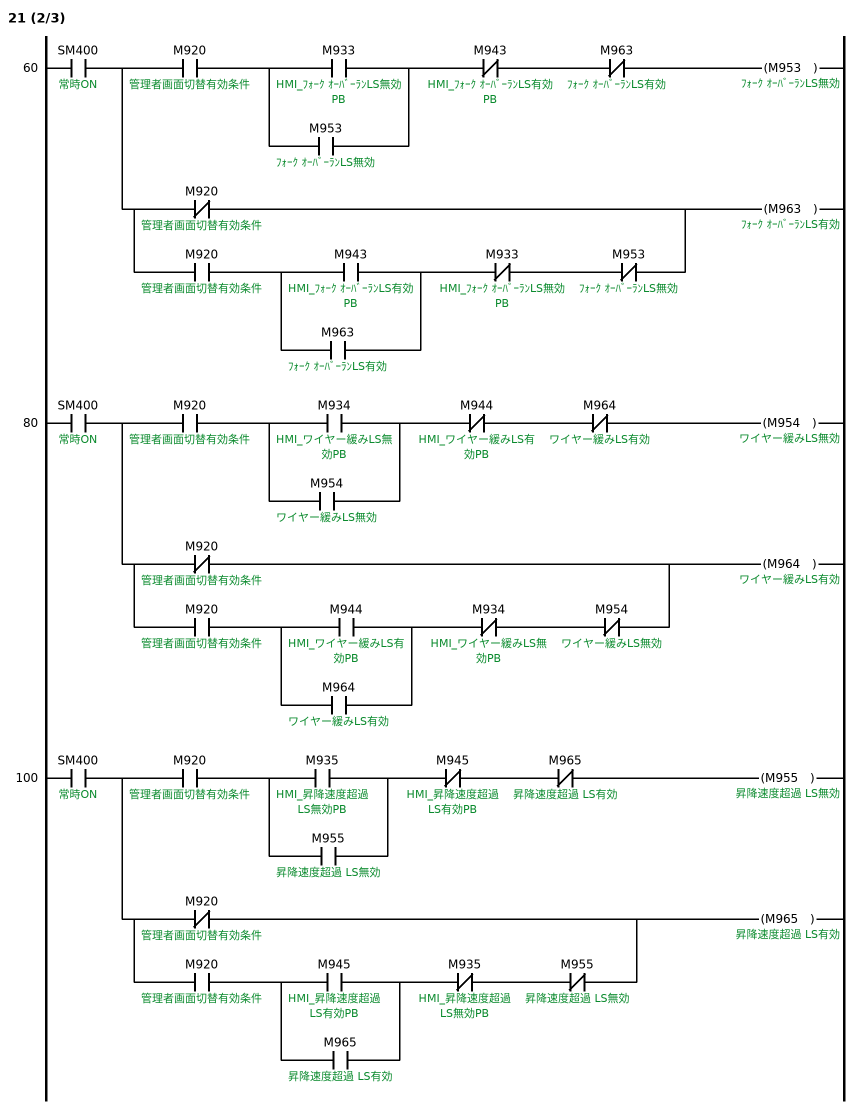
60    LD      SM400  ; 常時ON
      MPS
      AND     M920  ; 管理者画面切替有効条件
      LD      M933  ; HMI_ﾌｫｰｸ ｵｰﾊﾞｰﾗﾝLS無効PB
      OR      M953  ; ﾌｫｰｸ ｵｰﾊﾞｰﾗﾝLS無効
      ANB
      ANI     M943  ; HMI_ﾌｫｰｸ ｵｰﾊﾞｰﾗﾝLS有効PB
      ANI     M963  ; ﾌｫｰｸ ｵｰﾊﾞｰﾗﾝLS有効
      OUT     M953  ; ﾌｫｰｸ ｵｰﾊﾞｰﾗﾝLS無効
      MPP
      LDI     M920  ; 管理者画面切替有効条件
      LD      M920  ; 管理者画面切替有効条件
      LD      M943  ; HMI_ﾌｫｰｸ ｵｰﾊﾞｰﾗﾝLS有効PB
      OR      M963  ; ﾌｫｰｸ ｵｰﾊﾞｰﾗﾝLS有効
      ANB
      ANI     M933  ; HMI_ﾌｫｰｸ ｵｰﾊﾞｰﾗﾝLS無効PB
      ANI     M953  ; ﾌｫｰｸ ｵｰﾊﾞｰﾗﾝLS無効
      ORB
      ANB
      OUT     M963  ; ﾌｫｰｸ ｵｰﾊﾞｰﾗﾝLS有効
80    LD      SM400  ; 常時ON
      MPS
      AND     M920  ; 管理者画面切替有効条件
      LD      M934  ; HMI_ワイヤー緩みLS無効PB
      OR      M954  ; ワイヤー緩みLS無効
      ANB
      ANI     M944  ; HMI_ワイヤー緩みLS有効PB
      ANI     M964  ; ワイヤー緩みLS有効
      OUT     M954  ; ワイヤー緩みLS無効
      MPP
      LDI     M920  ; 管理者画面切替有効条件
      LD      M920  ; 管理者画面切替有効条件
      LD      M944  ; HMI_ワイヤー緩みLS有効PB
      OR      M964  ; ワイヤー緩みLS有効
      ANB
      ANI     M934  ; HMI_ワイヤー緩みLS無効PB
      ANI     M954  ; ワイヤー緩みLS無効
      ORB
      ANB
      OUT     M964  ; ワイヤー緩みLS有効
100   LD      SM400  ; 常時ON
      MPS
      AND     M920  ; 管理者画面切替有効条件
      LD      M935  ; HMI_昇降速度超過 LS無効PB
      OR      M955  ; 昇降速度超過 LS無効
      ANB
      ANI     M945  ; HMI_昇降速度超過 LS有効PB
      ANI     M965  ; 昇降速度超過 LS有効
      OUT     M955  ; 昇降速度超過 LS無効
      MPP
      LDI     M920  ; 管理者画面切替有効条件
      LD      M920  ; 管理者画面切替有効条件
      LD      M945  ; HMI_昇降速度超過 LS有効PB
      OR      M965  ; 昇降速度超過 LS有効
      ANB
      ANI     M935  ; HMI_昇降速度超過 LS無効PB
      ANI     M955  ; 昇降速度超過 LS無効
      ORB
      ANB
      OUT     M965  ; 昇降速度超過 LS有効
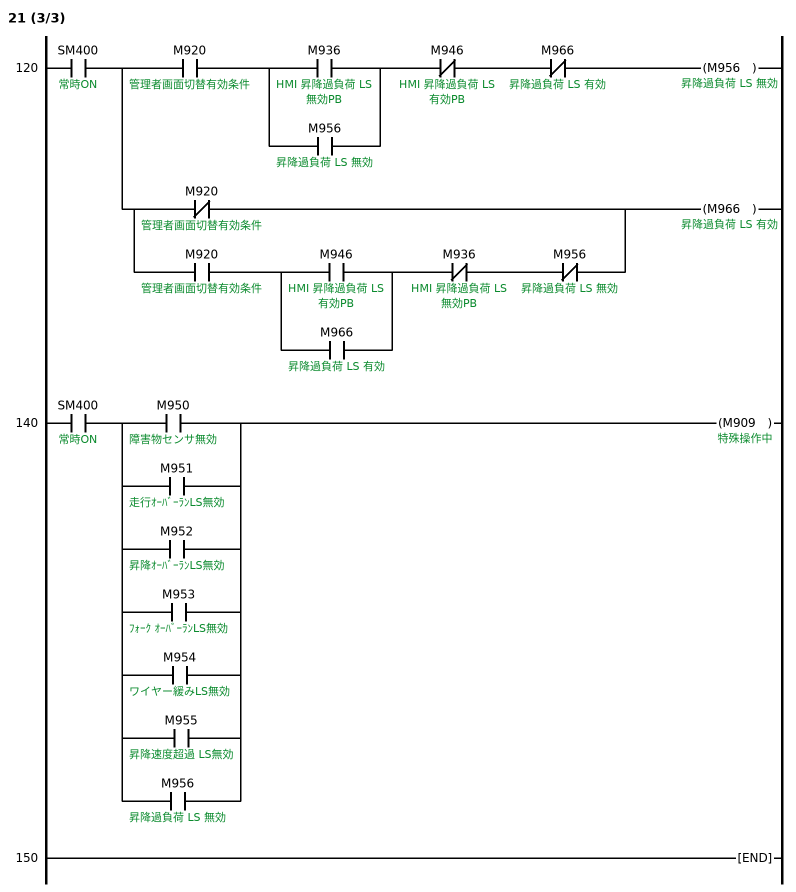
120   LD      SM400  ; 常時ON
      MPS
      AND     M920  ; 管理者画面切替有効条件
      LD      M936  ; HMI 昇降過負荷 LS 無効PB
      OR      M956  ; 昇降過負荷 LS 無効
      ANB
      ANI     M946  ; HMI 昇降過負荷 LS 有効PB
      ANI     M966  ; 昇降過負荷 LS 有効
      OUT     M956  ; 昇降過負荷 LS 無効
      MPP
      LDI     M920  ; 管理者画面切替有効条件
      LD      M920  ; 管理者画面切替有効条件
      LD      M946  ; HMI 昇降過負荷 LS 有効PB
      OR      M966  ; 昇降過負荷 LS 有効
      ANB
      ANI     M936  ; HMI 昇降過負荷 LS 無効PB
      ANI     M956  ; 昇降過負荷 LS 無効
      ORB
      ANB
      OUT     M966  ; 昇降過負荷 LS 有効
140   LD      SM400  ; 常時ON
      LD      M950  ; 障害物センサ無効
      OR      M951  ; 走行ｵｰﾊﾞｰﾗﾝLS無効
      OR      M952  ; 昇降ｵｰﾊﾞｰﾗﾝLS無効
      OR      M953  ; ﾌｫｰｸ ｵｰﾊﾞｰﾗﾝLS無効
      OR      M954  ; ワイヤー緩みLS無効
      OR      M955  ; 昇降速度超過 LS無効
      OR      M956  ; 昇降過負荷 LS 無効
      ANB
      OUT     M909  ; 特殊操作中
150   END
END_PROGRAM

PROGRAM 20  // 座標設定
VAR
  AO : INT;
  __IST_5190f969a590441b : I+ST_5190f969a590441b;
  __IST_28c7dc159632457c : I+ST_28c7dc159632457c;
  __IST_4e7308893d8d4cfe : I+ST_4e7308893d8d4cfe;
END_VAR
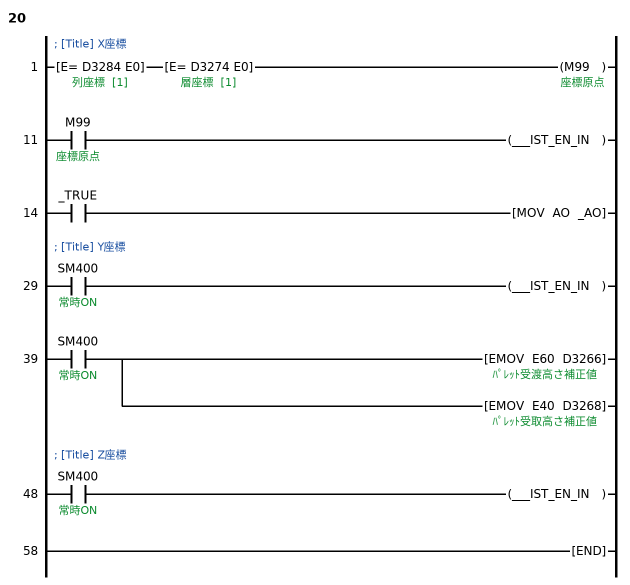
; [Title] X座標
1     LDE=    D3284 E0  ; 列座標  [1]
      ANDE=   D3274 E0  ; 層座標  [1]
      OUT     M99  ; 座標原点
; FB BLK START I+ST_5190f969a590441b(__IST_5190f969a590441b)
11    LD      M99  ; 座標原点
      OUT     ___IST_EN_IN
14    LD      _TRUE
      MOV     AO _AO
; FB START
; FB_NAME I+ST_5190f969a590441b
; INSTANCE_NAME __IST_5190f969a590441b
; FB IN_B:__IST_EN_IN
; FB OUT___IST_EN_OUT:B
; FB IN_W:AO
; FB OUT_AO:W
; FB END
; FB BLK END
; FB BLK START I+ST_28c7dc159632457c(__IST_28c7dc159632457c)
; [Title] Y座標
29    LD      SM400  ; 常時ON
      OUT     ___IST_EN_IN
; FB START
; FB_NAME I+ST_28c7dc159632457c
; INSTANCE_NAME __IST_28c7dc159632457c
; FB IN_B:__IST_EN_IN
; FB OUT___IST_EN_OUT:B
; FB END
; FB BLK END
39    LD      SM400  ; 常時ON
      EMOV    E60 D3266  ; ﾊﾟﾚｯﾄ受渡高さ補正値
      EMOV    E40 D3268  ; ﾊﾟﾚｯﾄ受取高さ補正値
; FB BLK START I+ST_4e7308893d8d4cfe(__IST_4e7308893d8d4cfe)
; [Title] Z座標
48    LD      SM400  ; 常時ON
      OUT     ___IST_EN_IN
; FB START
; FB_NAME I+ST_4e7308893d8d4cfe
; INSTANCE_NAME __IST_4e7308893d8d4cfe
; FB IN_B:__IST_EN_IN
; FB OUT___IST_EN_OUT:B
; FB END
; FB BLK END
58    END
END_PROGRAM

FUNCTION_BLOCK I+ST_5190f969a590441b
VAR_INPUT
  __IST_EN_IN : BOOL;
END_VAR
VAR_OUTPUT
  __IST_EN_OUT : BOOL;
END_VAR
VAR_IN_OUT
  AO : INT;
END_VAR
(* IST HEADER START *)
IF NOT __IST_EN_IN THEN __IST_EN_OUT:=FALSE; RETURN; END_IF;
(* VERSION=1:TYPE=STB *)
(* IST HEADER END *)
FOR AO:=1 TO 13 DO
	列座標[AO+1]:=列座標[AO] +1870.0;
END_FOR;
END_FUNCTION_BLOCK

FUNCTION_BLOCK I+ST_28c7dc159632457c
VAR_INPUT
  __IST_EN_IN : BOOL;
END_VAR
VAR_OUTPUT
  __IST_EN_OUT : BOOL;
END_VAR
(* IST HEADER START *)
IF NOT __IST_EN_IN THEN __IST_EN_OUT:=FALSE; RETURN; END_IF;
(* VERSION=1:TYPE=STB *)
(* IST HEADER END *)
層座標[1]:=0.0;
層座標[2]:=900.0;
層座標[3]:=1800.0;
層座標[4]:=2925.0;
層座標[5]:=3825.0;
END_FUNCTION_BLOCK

FUNCTION_BLOCK I+ST_4e7308893d8d4cfe
VAR_INPUT
  __IST_EN_IN : BOOL;
END_VAR
VAR_OUTPUT
  __IST_EN_OUT : BOOL;
END_VAR
(* IST HEADER START *)
IF NOT __IST_EN_IN THEN __IST_EN_OUT:=FALSE; RETURN; END_IF;
(* VERSION=1:TYPE=STB *)
(* IST HEADER END *)
Z座標[1]:=-1970.0;
Z座標[2]:=1970.0;
END_FUNCTION_BLOCK

PROGRAM 11  // Stackerフロー
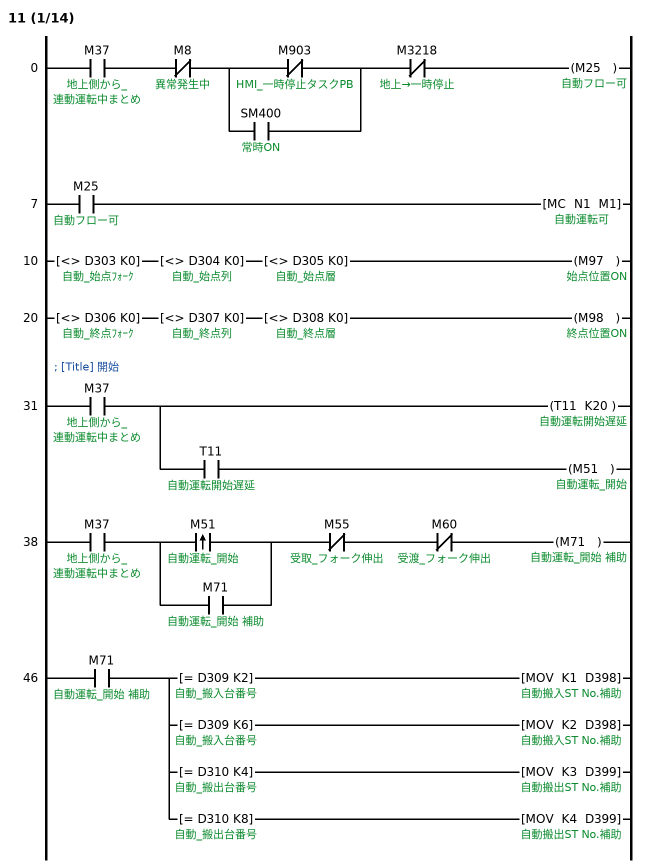
0     LD      M37  ; 地上側から_連動運転中まとめ
      ANI     M8  ; 異常発生中
      LDI     M903  ; HMI_一時停止タスクPB
      OR      SM400  ; 常時ON
      ANB
      ANI     M3218  ; 地上→一時停止
      OUT     M25  ; 自動フロー可
7     LD      M25  ; 自動フロー可
      MC      N1 M1  ; 自動運転可
10    LD<>    D303 K0  ; 自動_始点ﾌｫｰｸ
      AND<>   D304 K0  ; 自動_始点列
      AND<>   D305 K0  ; 自動_始点層
      OUT     M97  ; 始点位置ON
20    LD<>    D306 K0  ; 自動_終点ﾌｫｰｸ
      AND<>   D307 K0  ; 自動_終点列
      AND<>   D308 K0  ; 自動_終点層
      OUT     M98  ; 終点位置ON
; [Title] 開始
31    LD      M37  ; 地上側から_連動運転中まとめ
      OUT     T11 K20  ; 自動運転開始遅延
      AND     T11  ; 自動運転開始遅延
      OUT     M51  ; 自動運転_開始
38    LD      M37  ; 地上側から_連動運転中まとめ
      LDP     M51  ; 自動運転_開始
      OR      M71  ; 自動運転_開始 補助
      ANB
      ANI     M55  ; 受取_フォーク伸出
      ANI     M60  ; 受渡_フォーク伸出
      OUT     M71  ; 自動運転_開始 補助
46    LD      M71  ; 自動運転_開始 補助
      MPS
      AND=    D309 K2  ; 自動_搬入台番号
      MOV     K1 D398  ; 自動搬入ST No.補助
      MRD
      AND=    D309 K6  ; 自動_搬入台番号
      MOV     K2 D398
      MRD
      AND=    D310 K4  ; 自動_搬出台番号
      MOV     K3 D399  ; 自動搬出ST No.補助
      MPP
      AND=    D310 K8  ; 自動_搬出台番号
      MOV     K4 D399
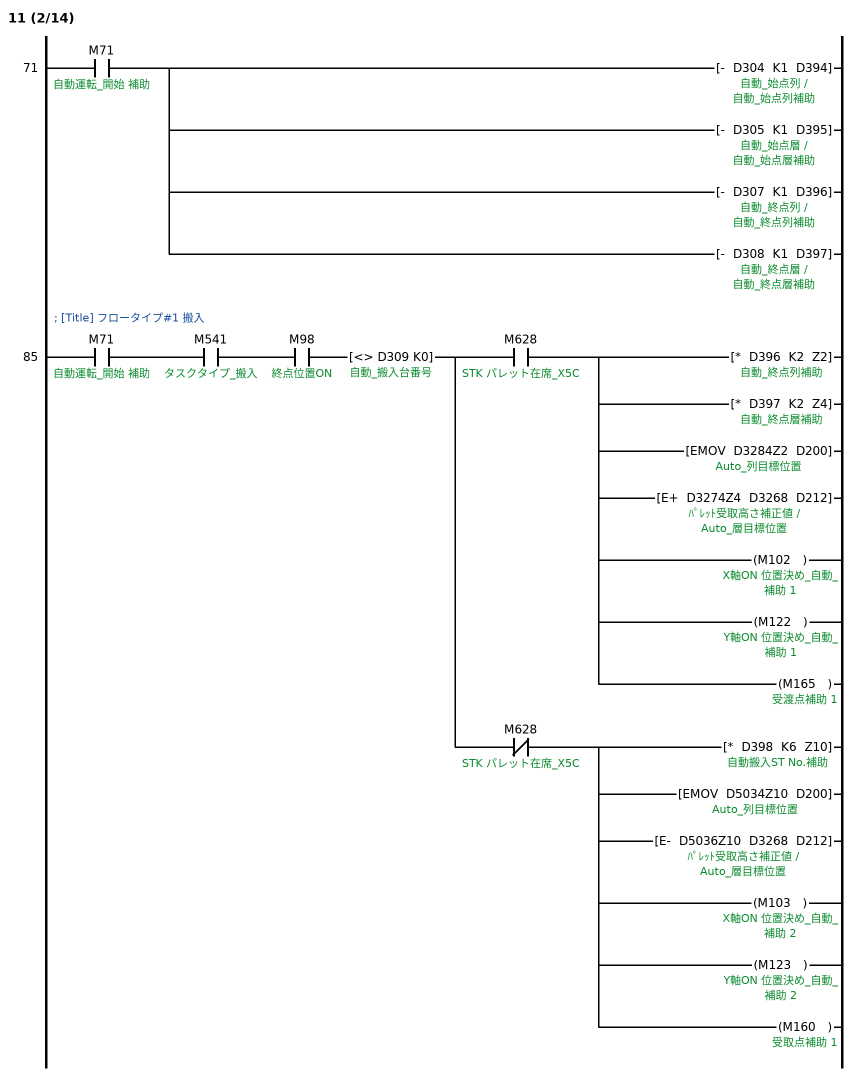
71    LD      M71  ; 自動運転_開始 補助
      -       D304 K1 D394  ; 自動_始点列補助
      -       D305 K1 D395  ; 自動_始点層補助
      -       D307 K1 D396  ; 自動_終点列補助
      -       D308 K1 D397  ; 自動_終点層補助
; [Title] フロータイプ#1 搬入
85    LD      M71  ; 自動運転_開始 補助
      AND     M541  ; タスクタイプ_搬入
      AND     M98  ; 終点位置ON
      AND<>   D309 K0  ; 自動_搬入台番号
      MPS
      AND     M628  ; STK パレット在席_X5C
      *       D396 K2 Z2
      *       D397 K2 Z4
      EMOV    D3284Z2 D200  ; Auto_列目標位置
      E+      D3274Z4 D3268 D212  ; ﾊﾟﾚｯﾄ受取高さ補正値 / Auto_層目標位置
      OUT     M102  ; X軸ON 位置決め_自動_補助 1
      OUT     M122  ; Y軸ON 位置決め_自動_補助 1
      OUT     M165  ; 受渡点補助 1
      MPP
      ANI     M628  ; STK パレット在席_X5C
      *       D398 K6 Z10
      EMOV    D5034Z10 D200
      E-      D5036Z10 D3268 D212
      OUT     M103  ; X軸ON 位置決め_自動_補助 2
      OUT     M123  ; Y軸ON 位置決め_自動_補助 2
      OUT     M160  ; 受取点補助 1
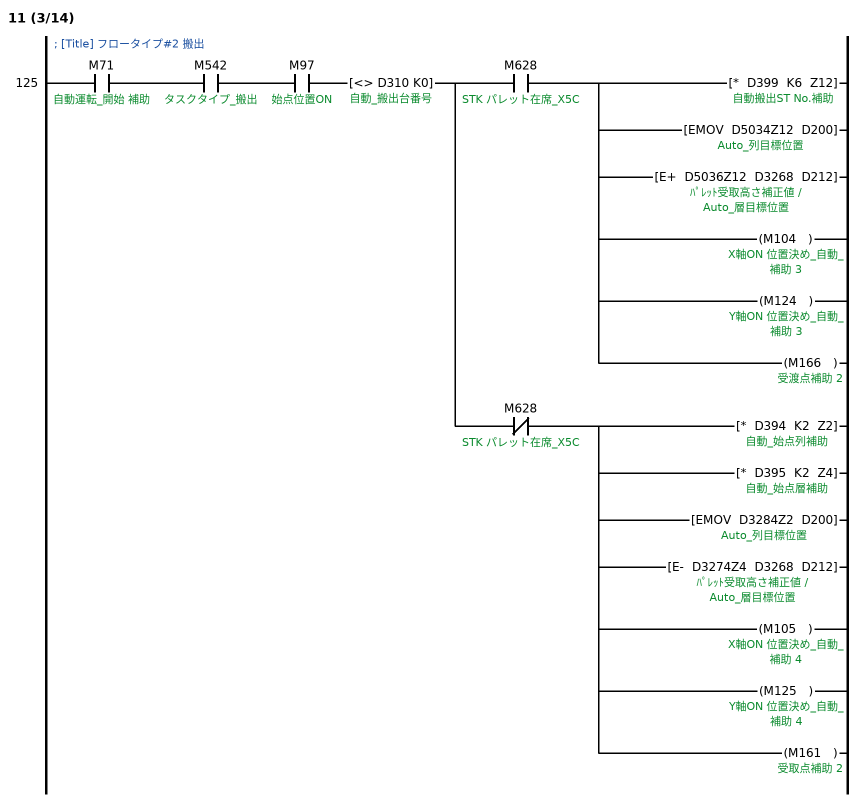
; [Title] フロータイプ#2 搬出
125   LD      M71  ; 自動運転_開始 補助
      AND     M542  ; タスクタイプ_搬出
      AND     M97  ; 始点位置ON
      AND<>   D310 K0  ; 自動_搬出台番号
      MPS
      AND     M628  ; STK パレット在席_X5C
      *       D399 K6 Z12
      EMOV    D5034Z12 D200
      E+      D5036Z12 D3268 D212
      OUT     M104  ; X軸ON 位置決め_自動_補助 3
      OUT     M124  ; Y軸ON 位置決め_自動_補助 3
      OUT     M166  ; 受渡点補助 2
      MPP
      ANI     M628  ; STK パレット在席_X5C
      *       D394 K2 Z2
      *       D395 K2 Z4
      EMOV    D3284Z2 D200
      E-      D3274Z4 D3268 D212
      OUT     M105  ; X軸ON 位置決め_自動_補助 4
      OUT     M125  ; Y軸ON 位置決め_自動_補助 4
      OUT     M161  ; 受取点補助 2
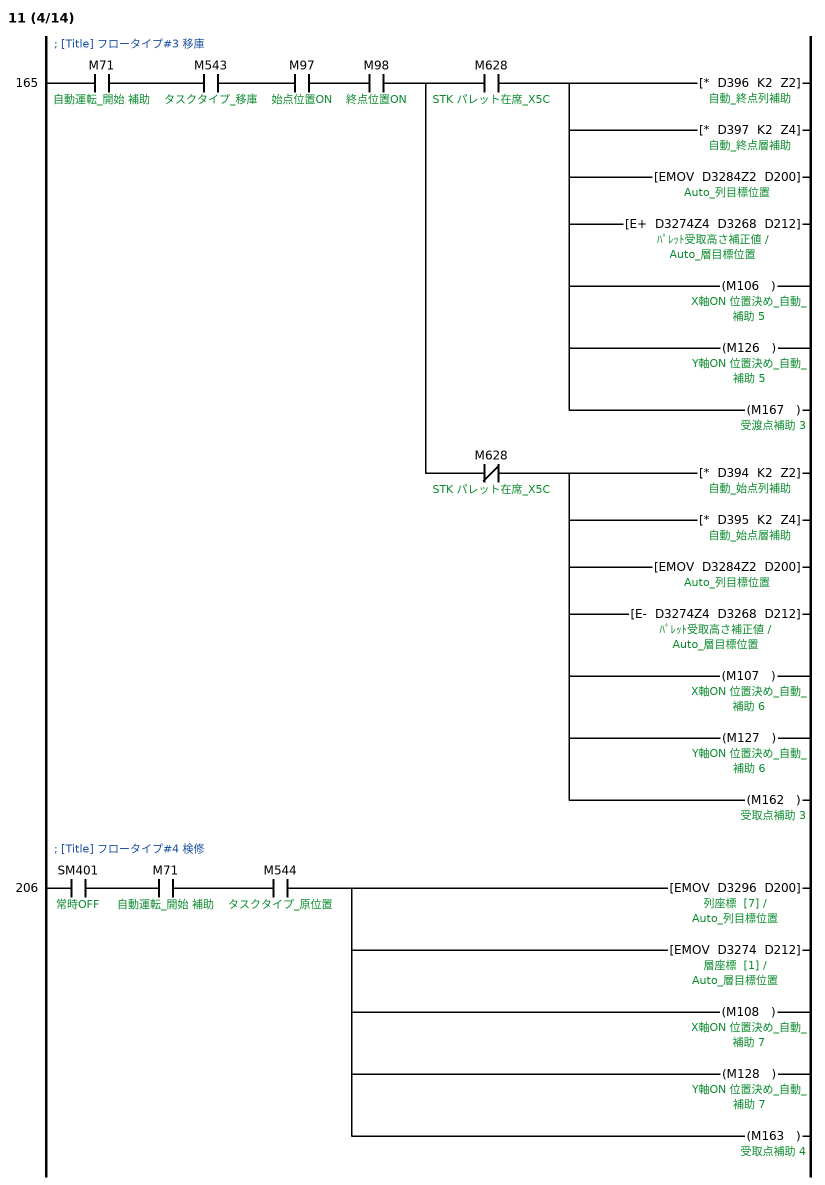
; [Title] フロータイプ#3 移庫
165   LD      M71  ; 自動運転_開始 補助
      AND     M543  ; タスクタイプ_移庫
      AND     M97  ; 始点位置ON
      AND     M98  ; 終点位置ON
      MPS
      AND     M628  ; STK パレット在席_X5C
      *       D396 K2 Z2
      *       D397 K2 Z4
      EMOV    D3284Z2 D200
      E+      D3274Z4 D3268 D212
      OUT     M106  ; X軸ON 位置決め_自動_補助 5
      OUT     M126  ; Y軸ON 位置決め_自動_補助 5
      OUT     M167  ; 受渡点補助 3
      MPP
      ANI     M628  ; STK パレット在席_X5C
      *       D394 K2 Z2
      *       D395 K2 Z4
      EMOV    D3284Z2 D200
      E-      D3274Z4 D3268 D212
      OUT     M107  ; X軸ON 位置決め_自動_補助 6
      OUT     M127  ; Y軸ON 位置決め_自動_補助 6
      OUT     M162  ; 受取点補助 3
; [Title] フロータイプ#4 検修
206   LD      SM401  ; 常時OFF
      AND     M71  ; 自動運転_開始 補助
      AND     M544  ; タスクタイプ_原位置
      EMOV    D3296 D200  ; 列座標  [7]
      EMOV    D3274 D212  ; 層座標  [1]
      OUT     M108  ; X軸ON 位置決め_自動_補助 7
      OUT     M128  ; Y軸ON 位置決め_自動_補助 7
      OUT     M163  ; 受取点補助 4
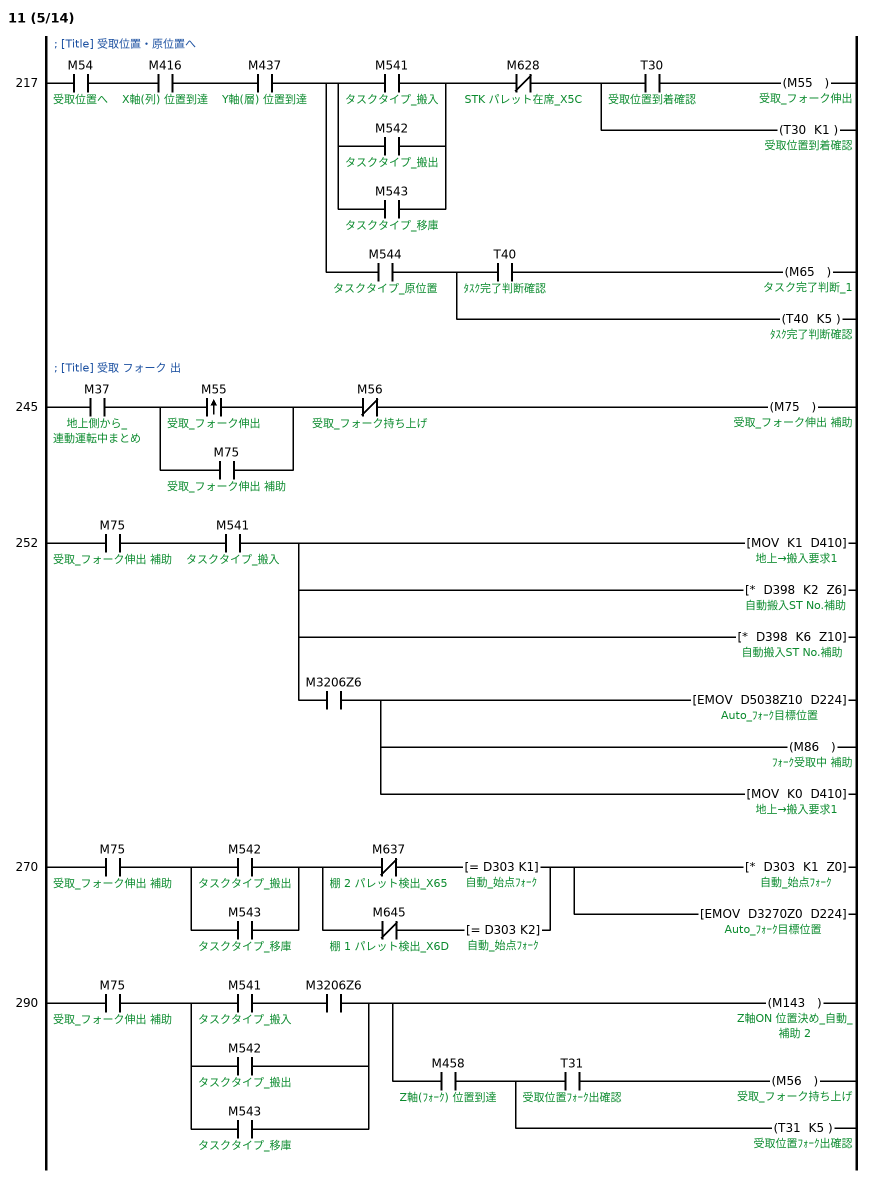
; [Title] 受取位置・原位置へ
217   LD      M54  ; 受取位置へ
      AND     M416  ; X軸(列) 位置到達
      AND     M437  ; Y軸(層) 位置到達
      MPS
      LD      M541  ; タスクタイプ_搬入
      OR      M542  ; タスクタイプ_搬出
      OR      M543  ; タスクタイプ_移庫
      ANB
      ANI     M628  ; STK パレット在席_X5C
      MPS
      AND     T30  ; 受取位置到着確認
      OUT     M55  ; 受取_フォーク伸出
      MPP
      OUT     T30 K1  ; 受取位置到着確認
      MPP
      AND     M544  ; タスクタイプ_原位置
      MPS
      AND     T40  ; ﾀｽｸ完了判断確認
      OUT     M65  ; タスク完了判断_1
      MPP
      OUT     T40 K5  ; ﾀｽｸ完了判断確認
; [Title] 受取 フォーク 出
245   LD      M37  ; 地上側から_連動運転中まとめ
      LDP     M55  ; 受取_フォーク伸出
      OR      M75  ; 受取_フォーク伸出 補助
      ANB
      ANI     M56  ; 受取_フォーク持ち上げ
      OUT     M75  ; 受取_フォーク伸出 補助
252   LD      M75  ; 受取_フォーク伸出 補助
      AND     M541  ; タスクタイプ_搬入
      MOV     K1 D410  ; 地上→搬入要求1
      *       D398 K2 Z6
      *       D398 K6 Z10
      AND     M3206Z6
      EMOV    D5038Z10 D224  ; Auto_ﾌｫｰｸ目標位置
      OUT     M86  ; ﾌｫｰｸ受取中 補助
      MOV     K0 D410
270   LD      M75  ; 受取_フォーク伸出 補助
      LD      M542  ; タスクタイプ_搬出
      OR      M543  ; タスクタイプ_移庫
      ANB
      LDI     M637  ; 棚 2 パレット検出_X65
      AND=    D303 K1  ; 自動_始点ﾌｫｰｸ
      LDI     M645  ; 棚 1 パレット検出_X6D
      AND=    D303 K2  ; 自動_始点ﾌｫｰｸ
      ORB
      ANB
      *       D303 K1 Z0
      EMOV    D3270Z0 D224
290   LD      M75  ; 受取_フォーク伸出 補助
      LD      M541  ; タスクタイプ_搬入
      AND     M3206Z6
      OR      M542  ; タスクタイプ_搬出
      OR      M543  ; タスクタイプ_移庫
      ANB
      OUT     M143  ; Z軸ON 位置決め_自動_補助 2
      AND     M458  ; Z軸(ﾌｫｰｸ) 位置到達
      MPS
      AND     T31  ; 受取位置ﾌｫｰｸ出確認
      OUT     M56  ; 受取_フォーク持ち上げ
      MPP
      OUT     T31 K5  ; 受取位置ﾌｫｰｸ出確認
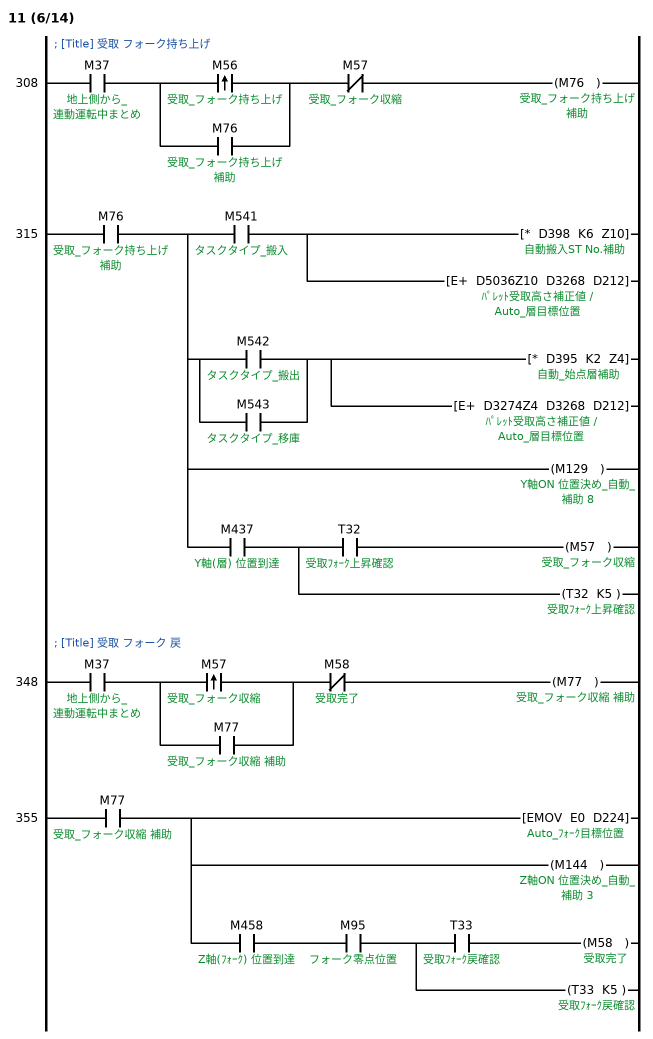
; [Title] 受取 フォーク持ち上げ
308   LD      M37  ; 地上側から_連動運転中まとめ
      LDP     M56  ; 受取_フォーク持ち上げ
      OR      M76  ; 受取_フォーク持ち上げ 補助
      ANB
      ANI     M57  ; 受取_フォーク収縮
      OUT     M76  ; 受取_フォーク持ち上げ 補助
315   LD      M76  ; 受取_フォーク持ち上げ 補助
      MPS
      AND     M541  ; タスクタイプ_搬入
      *       D398 K6 Z10
      E+      D5036Z10 D3268 D212
      MRD
      LD      M542  ; タスクタイプ_搬出
      OR      M543  ; タスクタイプ_移庫
      ANB
      *       D395 K2 Z4
      E+      D3274Z4 D3268 D212
      MPP
      OUT     M129  ; Y軸ON 位置決め_自動_補助 8
      AND     M437  ; Y軸(層) 位置到達
      MPS
      AND     T32  ; 受取ﾌｫｰｸ上昇確認
      OUT     M57  ; 受取_フォーク収縮
      MPP
      OUT     T32 K5  ; 受取ﾌｫｰｸ上昇確認
; [Title] 受取 フォーク 戻
348   LD      M37  ; 地上側から_連動運転中まとめ
      LDP     M57  ; 受取_フォーク収縮
      OR      M77  ; 受取_フォーク収縮 補助
      ANB
      ANI     M58  ; 受取完了
      OUT     M77  ; 受取_フォーク収縮 補助
355   LD      M77  ; 受取_フォーク収縮 補助
      EMOV    E0 D224
      OUT     M144  ; Z軸ON 位置決め_自動_補助 3
      AND     M458  ; Z軸(ﾌｫｰｸ) 位置到達
      AND     M95  ; フォーク零点位置
      MPS
      AND     T33  ; 受取ﾌｫｰｸ戻確認
      OUT     M58  ; 受取完了
      MPP
      OUT     T33 K5  ; 受取ﾌｫｰｸ戻確認
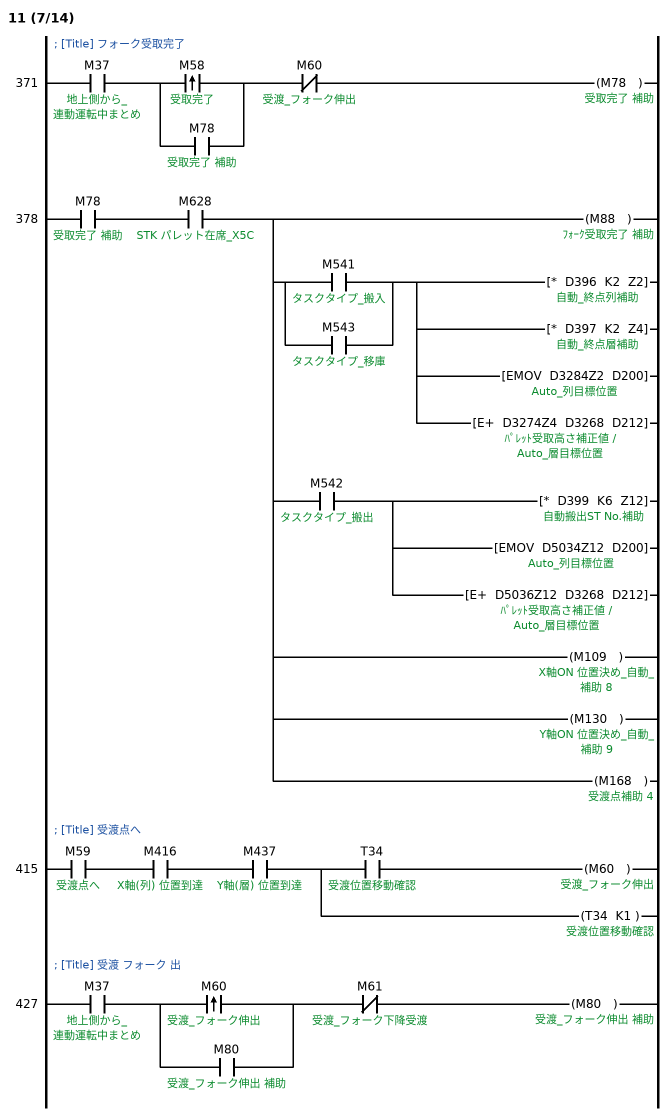
; [Title] フォーク受取完了
371   LD      M37  ; 地上側から_連動運転中まとめ
      LDP     M58  ; 受取完了
      OR      M78  ; 受取完了 補助
      ANB
      ANI     M60  ; 受渡_フォーク伸出
      OUT     M78  ; 受取完了 補助
378   LD      M78  ; 受取完了 補助
      AND     M628  ; STK パレット在席_X5C
      OUT     M88  ; ﾌｫｰｸ受取完了 補助
      MPS
      LD      M541  ; タスクタイプ_搬入
      OR      M543  ; タスクタイプ_移庫
      ANB
      *       D396 K2 Z2
      *       D397 K2 Z4
      EMOV    D3284Z2 D200
      E+      D3274Z4 D3268 D212
      MRD
      AND     M542  ; タスクタイプ_搬出
      *       D399 K6 Z12
      EMOV    D5034Z12 D200
      E+      D5036Z12 D3268 D212
      MPP
      OUT     M109  ; X軸ON 位置決め_自動_補助 8
      OUT     M130  ; Y軸ON 位置決め_自動_補助 9
      OUT     M168  ; 受渡点補助 4
; [Title] 受渡点へ
415   LD      M59  ; 受渡点へ
      AND     M416  ; X軸(列) 位置到達
      AND     M437  ; Y軸(層) 位置到達
      MPS
      AND     T34  ; 受渡位置移動確認
      OUT     M60  ; 受渡_フォーク伸出
      MPP
      OUT     T34 K1  ; 受渡位置移動確認
; [Title] 受渡 フォーク 出
427   LD      M37  ; 地上側から_連動運転中まとめ
      LDP     M60  ; 受渡_フォーク伸出
      OR      M80  ; 受渡_フォーク伸出 補助
      ANB
      ANI     M61  ; 受渡_フォーク下降受渡
      OUT     M80  ; 受渡_フォーク伸出 補助
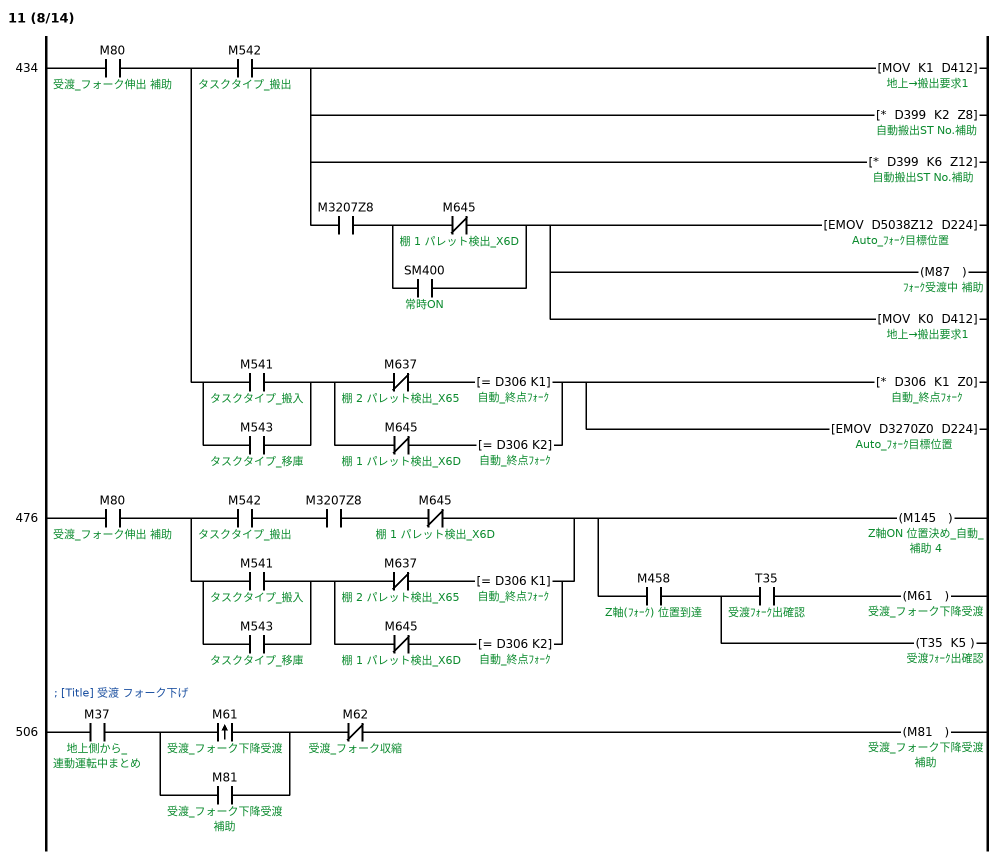
434   LD      M80  ; 受渡_フォーク伸出 補助
      MPS
      AND     M542  ; タスクタイプ_搬出
      MOV     K1 D412  ; 地上→搬出要求1
      *       D399 K2 Z8
      *       D399 K6 Z12
      AND     M3207Z8
      LDI     M645  ; 棚 1 パレット検出_X6D
      OR      SM400  ; 常時ON
      ANB
      EMOV    D5038Z12 D224
      OUT     M87  ; ﾌｫｰｸ受渡中 補助
      MOV     K0 D412
      MPP
      LD      M541  ; タスクタイプ_搬入
      OR      M543  ; タスクタイプ_移庫
      ANB
      LDI     M637  ; 棚 2 パレット検出_X65
      AND=    D306 K1  ; 自動_終点ﾌｫｰｸ
      LDI     M645  ; 棚 1 パレット検出_X6D
      AND=    D306 K2  ; 自動_終点ﾌｫｰｸ
      ORB
      ANB
      *       D306 K1 Z0
      EMOV    D3270Z0 D224
476   LD      M80  ; 受渡_フォーク伸出 補助
      LD      M542  ; タスクタイプ_搬出
      AND     M3207Z8
      ANI     M645  ; 棚 1 パレット検出_X6D
      LD      M541  ; タスクタイプ_搬入
      OR      M543  ; タスクタイプ_移庫
      LDI     M637  ; 棚 2 パレット検出_X65
      AND=    D306 K1  ; 自動_終点ﾌｫｰｸ
      LDI     M645  ; 棚 1 パレット検出_X6D
      AND=    D306 K2  ; 自動_終点ﾌｫｰｸ
      ORB
      ANB
      ORB
      ANB
      OUT     M145  ; Z軸ON 位置決め_自動_補助 4
      AND     M458  ; Z軸(ﾌｫｰｸ) 位置到達
      MPS
      AND     T35  ; 受渡ﾌｫｰｸ出確認
      OUT     M61  ; 受渡_フォーク下降受渡
      MPP
      OUT     T35 K5  ; 受渡ﾌｫｰｸ出確認
; [Title] 受渡 フォーク下げ
506   LD      M37  ; 地上側から_連動運転中まとめ
      LDP     M61  ; 受渡_フォーク下降受渡
      OR      M81  ; 受渡_フォーク下降受渡 補助
      ANB
      ANI     M62  ; 受渡_フォーク収縮
      OUT     M81  ; 受渡_フォーク下降受渡 補助
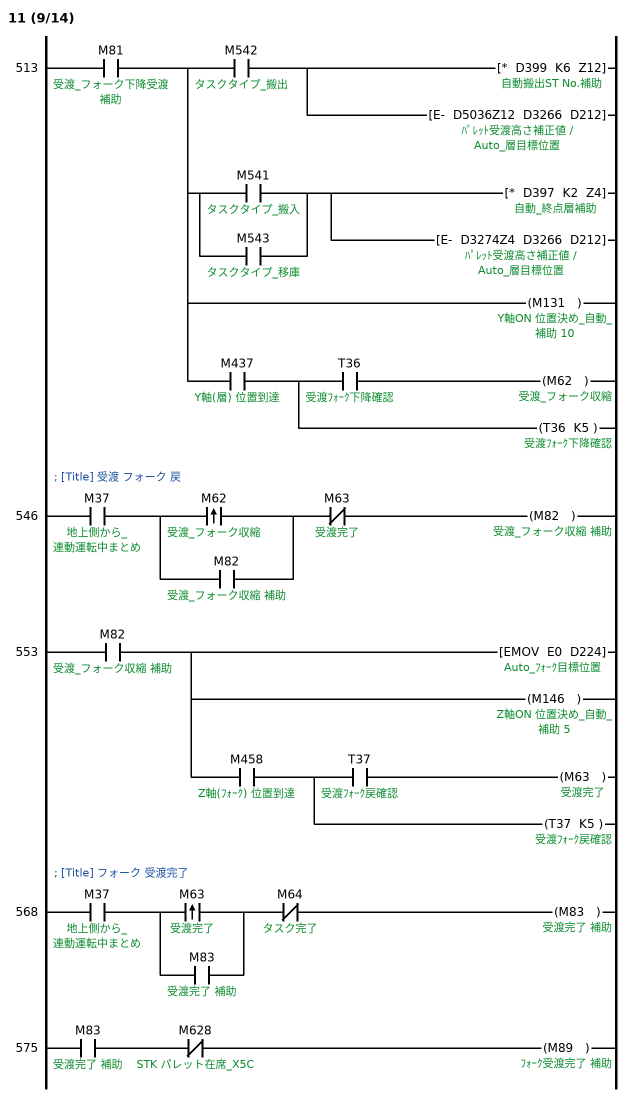
513   LD      M81  ; 受渡_フォーク下降受渡 補助
      MPS
      AND     M542  ; タスクタイプ_搬出
      *       D399 K6 Z12
      E-      D5036Z12 D3266 D212  ; ﾊﾟﾚｯﾄ受渡高さ補正値
      MRD
      LD      M541  ; タスクタイプ_搬入
      OR      M543  ; タスクタイプ_移庫
      ANB
      *       D397 K2 Z4
      E-      D3274Z4 D3266 D212
      MPP
      OUT     M131  ; Y軸ON 位置決め_自動_補助 10
      AND     M437  ; Y軸(層) 位置到達
      MPS
      AND     T36  ; 受渡ﾌｫｰｸ下降確認
      OUT     M62  ; 受渡_フォーク収縮
      MPP
      OUT     T36 K5  ; 受渡ﾌｫｰｸ下降確認
; [Title] 受渡 フォーク 戻
546   LD      M37  ; 地上側から_連動運転中まとめ
      LDP     M62  ; 受渡_フォーク収縮
      OR      M82  ; 受渡_フォーク収縮 補助
      ANB
      ANI     M63  ; 受渡完了
      OUT     M82  ; 受渡_フォーク収縮 補助
553   LD      M82  ; 受渡_フォーク収縮 補助
      EMOV    E0 D224
      OUT     M146  ; Z軸ON 位置決め_自動_補助 5
      AND     M458  ; Z軸(ﾌｫｰｸ) 位置到達
      MPS
      AND     T37  ; 受渡ﾌｫｰｸ戻確認
      OUT     M63  ; 受渡完了
      MPP
      OUT     T37 K5  ; 受渡ﾌｫｰｸ戻確認
; [Title] フォーク 受渡完了
568   LD      M37  ; 地上側から_連動運転中まとめ
      LDP     M63  ; 受渡完了
      OR      M83  ; 受渡完了 補助
      ANB
      ANI     M64  ; タスク完了
      OUT     M83  ; 受渡完了 補助
575   LD      M83  ; 受渡完了 補助
      ANI     M628  ; STK パレット在席_X5C
      OUT     M89  ; ﾌｫｰｸ受渡完了 補助
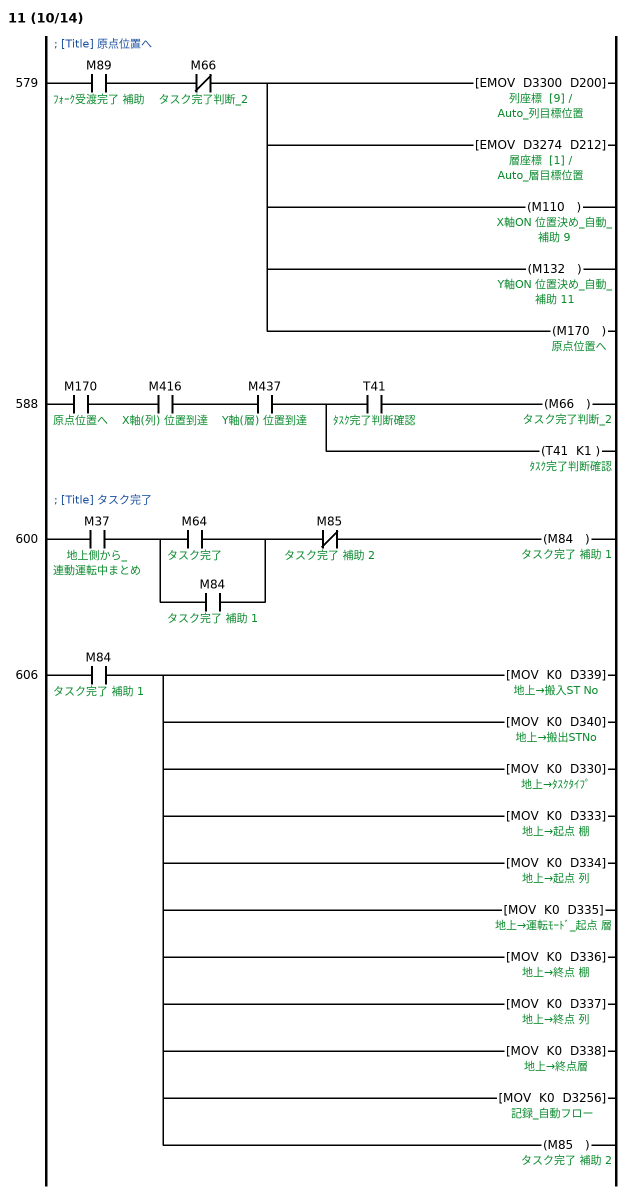
; [Title] 原点位置へ
579   LD      M89  ; ﾌｫｰｸ受渡完了 補助
      ANI     M66  ; タスク完了判断_2
      EMOV    D3300 D200  ; 列座標  [9]
      EMOV    D3274 D212
      OUT     M110  ; X軸ON 位置決め_自動_補助 9
      OUT     M132  ; Y軸ON 位置決め_自動_補助 11
      OUT     M170  ; 原点位置へ
588   LD      M170  ; 原点位置へ
      AND     M416  ; X軸(列) 位置到達
      AND     M437  ; Y軸(層) 位置到達
      MPS
      AND     T41  ; ﾀｽｸ完了判断確認
      OUT     M66  ; タスク完了判断_2
      MPP
      OUT     T41 K1  ; ﾀｽｸ完了判断確認
; [Title] タスク完了
600   LD      M37  ; 地上側から_連動運転中まとめ
      LD      M64  ; タスク完了
      OR      M84  ; タスク完了 補助 1
      ANB
      ANI     M85  ; タスク完了 補助 2
      OUT     M84  ; タスク完了 補助 1
606   LD      M84  ; タスク完了 補助 1
      MOV     K0 D339  ; 地上→搬入ST No
      MOV     K0 D340  ; 地上→搬出STNo
      MOV     K0 D330  ; 地上→ﾀｽｸﾀｲﾌﾟ
      MOV     K0 D333  ; 地上→起点 棚
      MOV     K0 D334  ; 地上→起点 列
      MOV     K0 D335  ; 地上→運転ﾓｰﾄﾞ_起点 層
      MOV     K0 D336  ; 地上→終点 棚
      MOV     K0 D337  ; 地上→終点 列
      MOV     K0 D338  ; 地上→終点層
      MOV     K0 D3256  ; 記録_自動フロー
      OUT     M85  ; タスク完了 補助 2
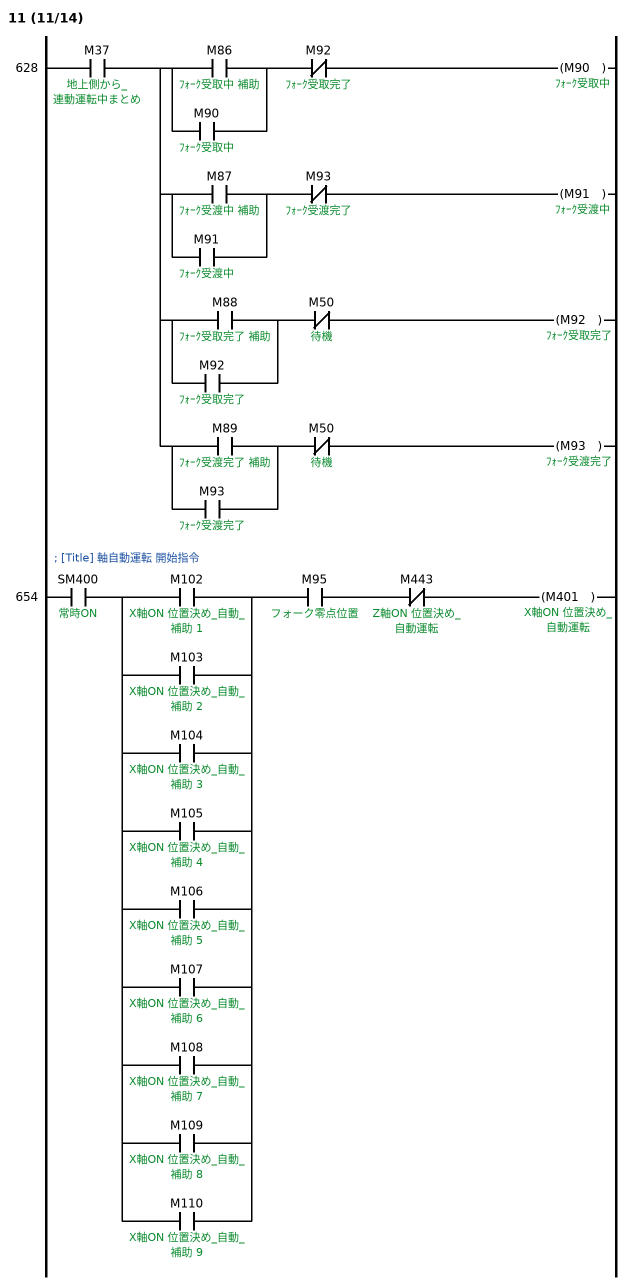
628   LD      M37  ; 地上側から_連動運転中まとめ
      MPS
      LD      M86  ; ﾌｫｰｸ受取中 補助
      OR      M90  ; ﾌｫｰｸ受取中
      ANB
      ANI     M92  ; ﾌｫｰｸ受取完了
      OUT     M90  ; ﾌｫｰｸ受取中
      MRD
      LD      M87  ; ﾌｫｰｸ受渡中 補助
      OR      M91  ; ﾌｫｰｸ受渡中
      ANB
      ANI     M93  ; ﾌｫｰｸ受渡完了
      OUT     M91  ; ﾌｫｰｸ受渡中
      MRD
      LD      M88  ; ﾌｫｰｸ受取完了 補助
      OR      M92  ; ﾌｫｰｸ受取完了
      ANB
      ANI     M50  ; 待機
      OUT     M92  ; ﾌｫｰｸ受取完了
      MPP
      LD      M89  ; ﾌｫｰｸ受渡完了 補助
      OR      M93  ; ﾌｫｰｸ受渡完了
      ANB
      ANI     M50  ; 待機
      OUT     M93  ; ﾌｫｰｸ受渡完了
; [Title] 軸自動運転 開始指令
654   LD      SM400  ; 常時ON
      LD      M102  ; X軸ON 位置決め_自動_補助 1
      OR      M103  ; X軸ON 位置決め_自動_補助 2
      OR      M104  ; X軸ON 位置決め_自動_補助 3
      OR      M105  ; X軸ON 位置決め_自動_補助 4
      OR      M106  ; X軸ON 位置決め_自動_補助 5
      OR      M107  ; X軸ON 位置決め_自動_補助 6
      OR      M108  ; X軸ON 位置決め_自動_補助 7
      OR      M109  ; X軸ON 位置決め_自動_補助 8
      OR      M110  ; X軸ON 位置決め_自動_補助 9
      ANB
      AND     M95  ; フォーク零点位置
      ANI     M443  ; Z軸ON 位置決め_自動運転
      OUT     M401  ; X軸ON 位置決め_自動運転
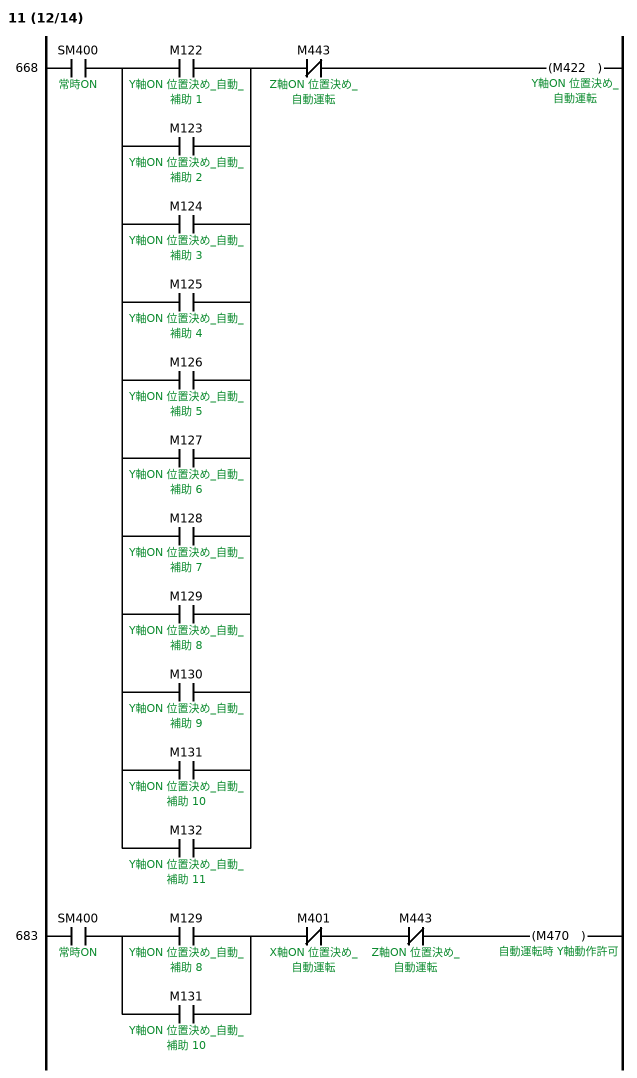
668   LD      SM400  ; 常時ON
      LD      M122  ; Y軸ON 位置決め_自動_補助 1
      OR      M123  ; Y軸ON 位置決め_自動_補助 2
      OR      M124  ; Y軸ON 位置決め_自動_補助 3
      OR      M125  ; Y軸ON 位置決め_自動_補助 4
      OR      M126  ; Y軸ON 位置決め_自動_補助 5
      OR      M127  ; Y軸ON 位置決め_自動_補助 6
      OR      M128  ; Y軸ON 位置決め_自動_補助 7
      OR      M129  ; Y軸ON 位置決め_自動_補助 8
      OR      M130  ; Y軸ON 位置決め_自動_補助 9
      OR      M131  ; Y軸ON 位置決め_自動_補助 10
      OR      M132  ; Y軸ON 位置決め_自動_補助 11
      ANB
      ANI     M443  ; Z軸ON 位置決め_自動運転
      OUT     M422  ; Y軸ON 位置決め_自動運転
683   LD      SM400  ; 常時ON
      LD      M129  ; Y軸ON 位置決め_自動_補助 8
      OR      M131  ; Y軸ON 位置決め_自動_補助 10
      ANB
      ANI     M401  ; X軸ON 位置決め_自動運転
      ANI     M443  ; Z軸ON 位置決め_自動運転
      OUT     M470  ; 自動運転時 Y軸動作許可
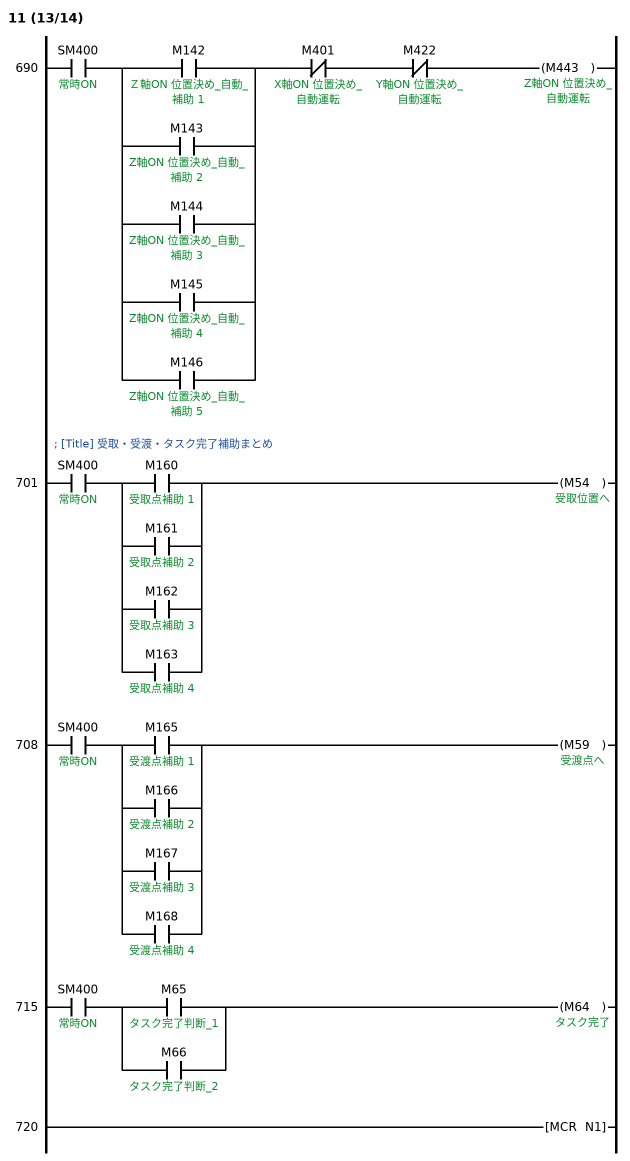
690   LD      SM400  ; 常時ON
      LD      M142  ; Ｚ軸ON 位置決め_自動_補助 1
      OR      M143  ; Z軸ON 位置決め_自動_補助 2
      OR      M144  ; Z軸ON 位置決め_自動_補助 3
      OR      M145  ; Z軸ON 位置決め_自動_補助 4
      OR      M146  ; Z軸ON 位置決め_自動_補助 5
      ANB
      ANI     M401  ; X軸ON 位置決め_自動運転
      ANI     M422  ; Y軸ON 位置決め_自動運転
      OUT     M443  ; Z軸ON 位置決め_自動運転
; [Title] 受取・受渡・タスク完了補助まとめ
701   LD      SM400  ; 常時ON
      LD      M160  ; 受取点補助 1
      OR      M161  ; 受取点補助 2
      OR      M162  ; 受取点補助 3
      OR      M163  ; 受取点補助 4
      ANB
      OUT     M54  ; 受取位置へ
708   LD      SM400  ; 常時ON
      LD      M165  ; 受渡点補助 1
      OR      M166  ; 受渡点補助 2
      OR      M167  ; 受渡点補助 3
      OR      M168  ; 受渡点補助 4
      ANB
      OUT     M59  ; 受渡点へ
715   LD      SM400  ; 常時ON
      LD      M65  ; タスク完了判断_1
      OR      M66  ; タスク完了判断_2
      ANB
      OUT     M64  ; タスク完了
720   MCR     N1
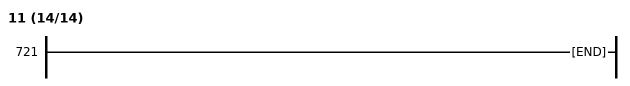
721   END
END_PROGRAM

FUNCTION_BLOCK I+ST_24fe211bdc5e490f
VAR_INPUT
  __IST_EN_IN : BOOL;
END_VAR
VAR_OUTPUT
  __IST_EN_OUT : BOOL;
END_VAR
VAR_IN_OUT
  AO1 : INT;
END_VAR
(* IST HEADER START *)
IF NOT __IST_EN_IN THEN __IST_EN_OUT:=FALSE; RETURN; END_IF;
(* VERSION=1:TYPE=STB *)
(* IST HEADER END *)
現在位置列:=0;
AO1:=0;
FOR AO1:=0 TO 14 DO
	IF Auto_Data.X軸現在位置 >(列座標[AO1]-50.0) AND Auto_Data.X軸現在位置 <(列座標[AO1]+50.0) THEN
	     現在位置列:=AO1;
		 EXIT;
	END_IF;
END_FOR;
END_FUNCTION_BLOCK

FUNCTION_BLOCK I+ST_2ed1eb90aebe4c54
VAR_INPUT
  __IST_EN_IN : BOOL;
END_VAR
VAR_OUTPUT
  __IST_EN_OUT : BOOL;
END_VAR
VAR_IN_OUT
  AO2 : INT;
END_VAR
(* IST HEADER START *)
IF NOT __IST_EN_IN THEN __IST_EN_OUT:=FALSE; RETURN; END_IF;
(* VERSION=1:TYPE=STB *)
(* IST HEADER END *)
現在位置層:=0;
AO2:=0;
FOR AO2:=0 TO 5 DO
	IF Auto_Data.Y軸現在位置 >(層座標[AO2]-50.0) AND Auto_Data.Y軸現在位置 <(層座標[AO2]+70.0) THEN
		現在位置層:=AO2;
		EXIT;
	END_IF;
END_FOR;
END_FUNCTION_BLOCK

PROGRAM 02  // Ether 入力 地上側盤
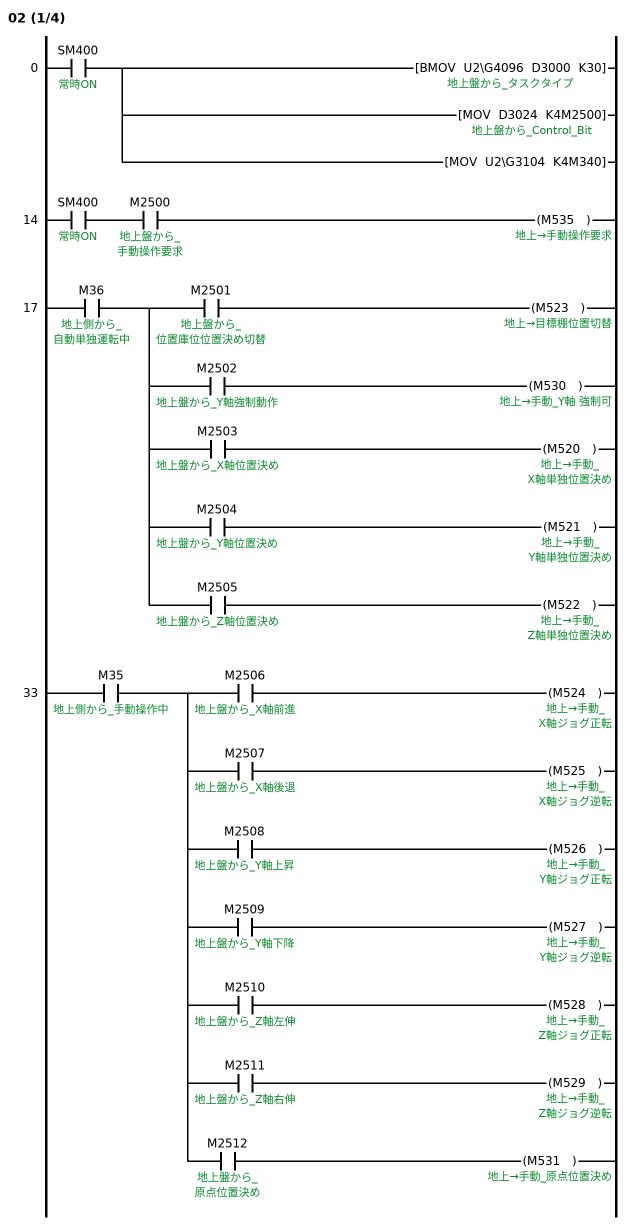
0     LD      SM400  ; 常時ON
      BMOV    U2\G4096 D3000 K30  ; 地上盤から_タスクタイプ
      MOV     D3024 K4M2500  ; 地上盤から_Control_Bit / 地上盤から_手動操作要求
      MOV     U2\G3104 K4M340  ; U2_通信異常
14    LD      SM400  ; 常時ON
      AND     M2500  ; 地上盤から_手動操作要求
      OUT     M535  ; 地上→手動操作要求
17    LD      M36  ; 地上側から_自動単独運転中
      MPS
      AND     M2501  ; 地上盤から_位置庫位位置決め切替
      OUT     M523  ; 地上→目標棚位置切替
      MRD
      AND     M2502  ; 地上盤から_Y軸強制動作
      OUT     M530  ; 地上→手動_Y軸 強制可
      MRD
      AND     M2503  ; 地上盤から_X軸位置決め
      OUT     M520  ; 地上→手動_X軸単独位置決め
      MRD
      AND     M2504  ; 地上盤から_Y軸位置決め
      OUT     M521  ; 地上→手動_Y軸単独位置決め
      MPP
      AND     M2505  ; 地上盤から_Z軸位置決め
      OUT     M522  ; 地上→手動_Z軸単独位置決め
33    LD      M35  ; 地上側から_手動操作中
      MPS
      AND     M2506  ; 地上盤から_X軸前進
      OUT     M524  ; 地上→手動_X軸ジョグ正転
      MRD
      AND     M2507  ; 地上盤から_X軸後退
      OUT     M525  ; 地上→手動_X軸ジョグ逆転
      MRD
      AND     M2508  ; 地上盤から_Y軸上昇
      OUT     M526  ; 地上→手動_Y軸ジョグ正転
      MRD
      AND     M2509  ; 地上盤から_Y軸下降
      OUT     M527  ; 地上→手動_Y軸ジョグ逆転
      MRD
      AND     M2510  ; 地上盤から_Z軸左伸
      OUT     M528  ; 地上→手動_Z軸ジョグ正転
      MRD
      AND     M2511  ; 地上盤から_Z軸右伸
      OUT     M529  ; 地上→手動_Z軸ジョグ逆転
      MPP
      AND     M2512  ; 地上盤から_原点位置決め
      OUT     M531  ; 地上→手動_原点位置決め
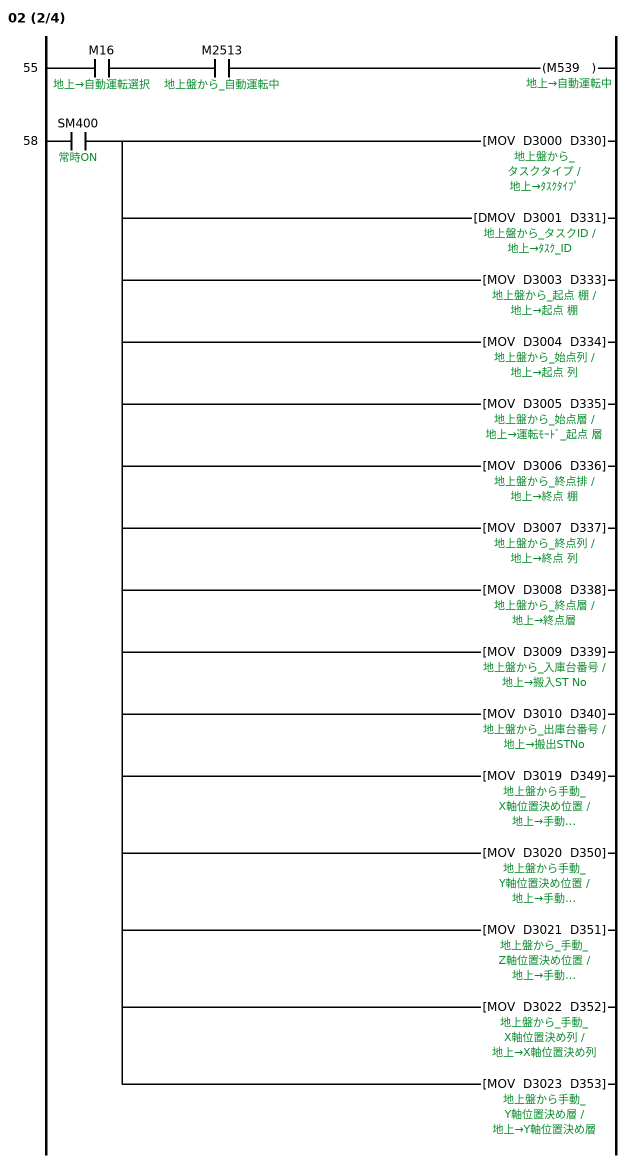
55    LD      M16  ; 地上→自動運転選択
      AND     M2513  ; 地上盤から_自動運転中
      OUT     M539  ; 地上→自動運転中
58    LD      SM400  ; 常時ON
      MOV     D3000 D330  ; 地上→ﾀｽｸﾀｲﾌﾟ
      DMOV    D3001 D331  ; 地上盤から_タスクID / 地上→ﾀｽｸ_ID
      MOV     D3003 D333  ; 地上盤から_起点 棚 / 地上→起点 棚
      MOV     D3004 D334  ; 地上盤から_始点列 / 地上→起点 列
      MOV     D3005 D335  ; 地上盤から_始点層 / 地上→運転ﾓｰﾄﾞ_起点 層
      MOV     D3006 D336  ; 地上盤から_終点排 / 地上→終点 棚
      MOV     D3007 D337  ; 地上盤から_終点列 / 地上→終点 列
      MOV     D3008 D338  ; 地上盤から_終点層 / 地上→終点層
      MOV     D3009 D339  ; 地上盤から_入庫台番号 / 地上→搬入ST No
      MOV     D3010 D340  ; 地上盤から_出庫台番号 / 地上→搬出STNo
      MOV     D3019 D349  ; 地上盤から手動_X軸位置決め位置 / 地上→手動_X軸位置決め座標
      MOV     D3020 D350  ; 地上盤から手動_Y軸位置決め位置 / 地上→手動_Y軸位置決め座標
      MOV     D3021 D351  ; 地上盤から_手動_Z軸位置決め位置 / 地上→手動_Z軸位置決め座標
      MOV     D3022 D352  ; 地上盤から_手動_X軸位置決め列 / 地上→X軸位置決め列
      MOV     D3023 D353  ; 地上盤から手動_Y軸位置決め層 / 地上→Y軸位置決め層
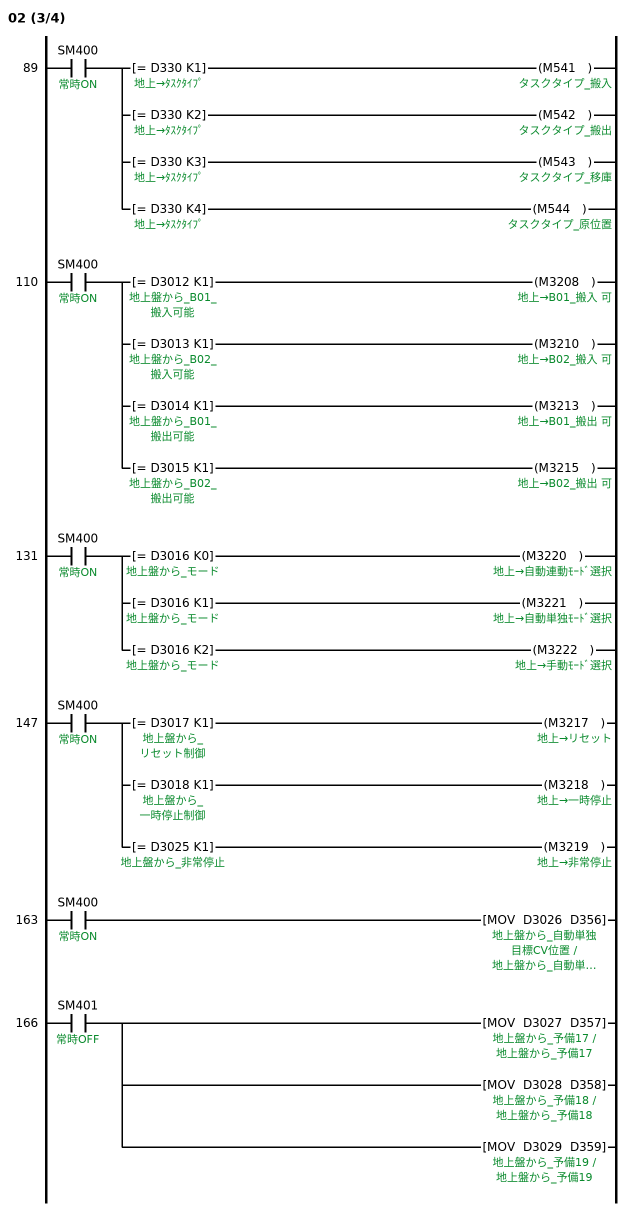
89    LD      SM400  ; 常時ON
      MPS
      AND=    D330 K1  ; 地上→ﾀｽｸﾀｲﾌﾟ
      OUT     M541  ; タスクタイプ_搬入
      MRD
      AND=    D330 K2  ; 地上→ﾀｽｸﾀｲﾌﾟ
      OUT     M542  ; タスクタイプ_搬出
      MRD
      AND=    D330 K3  ; 地上→ﾀｽｸﾀｲﾌﾟ
      OUT     M543  ; タスクタイプ_移庫
      MPP
      AND=    D330 K4  ; 地上→ﾀｽｸﾀｲﾌﾟ
      OUT     M544  ; タスクタイプ_原位置
110   LD      SM400  ; 常時ON
      MPS
      AND=    D3012 K1  ; 地上盤から_B01_搬入可能
      OUT     M3208  ; 地上→B01_搬入 可
      MRD
      AND=    D3013 K1  ; 地上盤から_B02_搬入可能
      OUT     M3210  ; 地上→B02_搬入 可
      MRD
      AND=    D3014 K1  ; 地上盤から_B01_搬出可能
      OUT     M3213  ; 地上→B01_搬出 可
      MPP
      AND=    D3015 K1  ; 地上盤から_B02_搬出可能
      OUT     M3215  ; 地上→B02_搬出 可
131   LD      SM400  ; 常時ON
      MPS
      AND=    D3016 K0  ; 地上盤から_モード
      OUT     M3220  ; 地上→自動連動ﾓｰﾄﾞ選択
      MRD
      AND=    D3016 K1  ; 地上盤から_モード
      OUT     M3221  ; 地上→自動単独ﾓｰﾄﾞ選択
      MPP
      AND=    D3016 K2  ; 地上盤から_モード
      OUT     M3222  ; 地上→手動ﾓｰﾄﾞ選択
147   LD      SM400  ; 常時ON
      MPS
      AND=    D3017 K1  ; 地上盤から_リセット制御
      OUT     M3217  ; 地上→リセット
      MRD
      AND=    D3018 K1  ; 地上盤から_一時停止制御
      OUT     M3218  ; 地上→一時停止
      MPP
      AND=    D3025 K1  ; 地上盤から_非常停止
      OUT     M3219  ; 地上→非常停止
163   LD      SM400  ; 常時ON
      MOV     D3026 D356  ; 地上盤から_自動単独 目標CV位置 / 地上盤から_自動単独 目標CV位置
166   LD      SM401  ; 常時OFF
      MOV     D3027 D357  ; 地上盤から_予備17 / 地上盤から_予備17
      MOV     D3028 D358  ; 地上盤から_予備18 / 地上盤から_予備18
      MOV     D3029 D359  ; 地上盤から_予備19 / 地上盤から_予備19
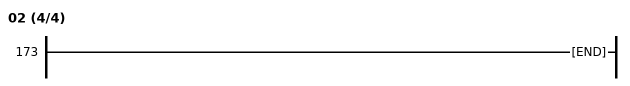
173   END
END_PROGRAM

PROGRAM 03  // Ether 入力 SEW INV
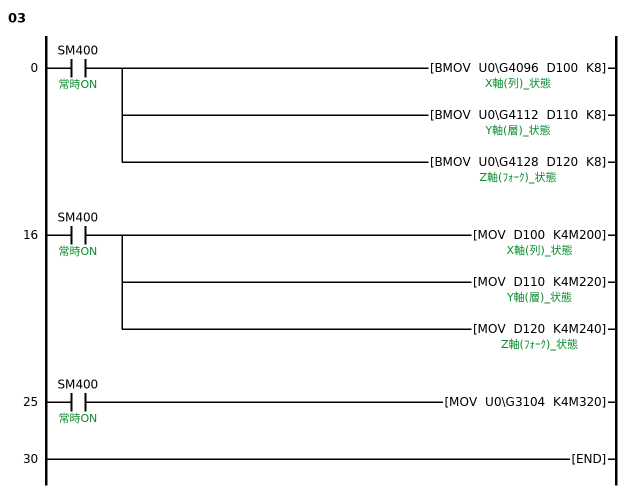
0     LD      SM400  ; 常時ON
      BMOV    U0\G4096 D100 K8  ; X軸(列)_状態
      BMOV    U0\G4112 D110 K8  ; Y軸(層)_状態
      BMOV    U0\G4128 D120 K8  ; Z軸(ﾌｫｰｸ)_状態
16    LD      SM400  ; 常時ON
      MOV     D100 K4M200  ; X軸_運転レディ
      MOV     D110 K4M220  ; Y軸_運転レディ
      MOV     D120 K4M240  ; Z軸_運転レディ
25    LD      SM400  ; 常時ON
      MOV     U0\G3104 K4M320  ; U0_X軸通信異常
30    END
END_PROGRAM

PROGRAM 51  // Ether 出力 地上側盤
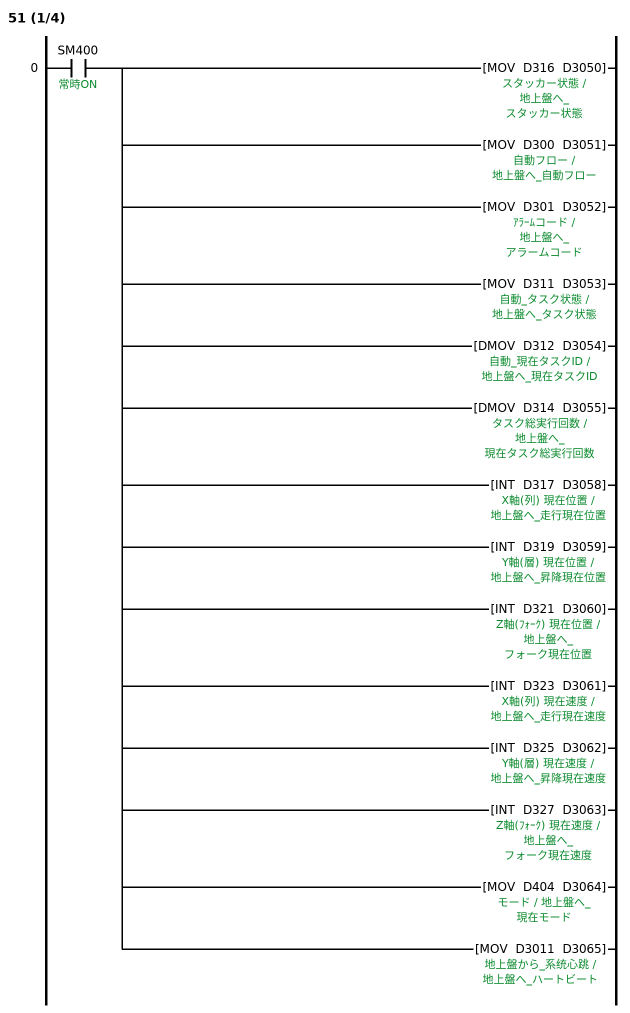
0     LD      SM400  ; 常時ON
      MOV     D316 D3050  ; スタッカー状態 / 地上盤へ_スタッカー状態
      MOV     D300 D3051  ; 自動フロー / 地上盤へ_自動フロー
      MOV     D301 D3052  ; ｱﾗｰﾑコード / 地上盤へ_アラームコード
      MOV     D311 D3053  ; 自動_タスク状態 / 地上盤へ_タスク状態
      DMOV    D312 D3054  ; 自動_現在タスクID / 地上盤へ_現在タスクID
      DMOV    D314 D3055  ; タスク総実行回数 / 地上盤へ_現在タスク総実行回数
      INT     D317 D3058  ; X軸(列) 現在位置 / 地上盤へ_走行現在位置
      INT     D319 D3059  ; Y軸(層) 現在位置 / 地上盤へ_昇降現在位置
      INT     D321 D3060  ; Z軸(ﾌｫｰｸ) 現在位置 / 地上盤へ_フォーク現在位置
      INT     D323 D3061  ; X軸(列) 現在速度 / 地上盤へ_走行現在速度
      INT     D325 D3062  ; Y軸(層) 現在速度 / 地上盤へ_昇降現在速度
      INT     D327 D3063  ; Z軸(ﾌｫｰｸ) 現在速度 / 地上盤へ_フォーク現在速度
      MOV     D404 D3064  ; モード / 地上盤へ_現在モード
      MOV     D3011 D3065  ; 地上盤から_系统心跳 / 地上盤へ_ハートビート
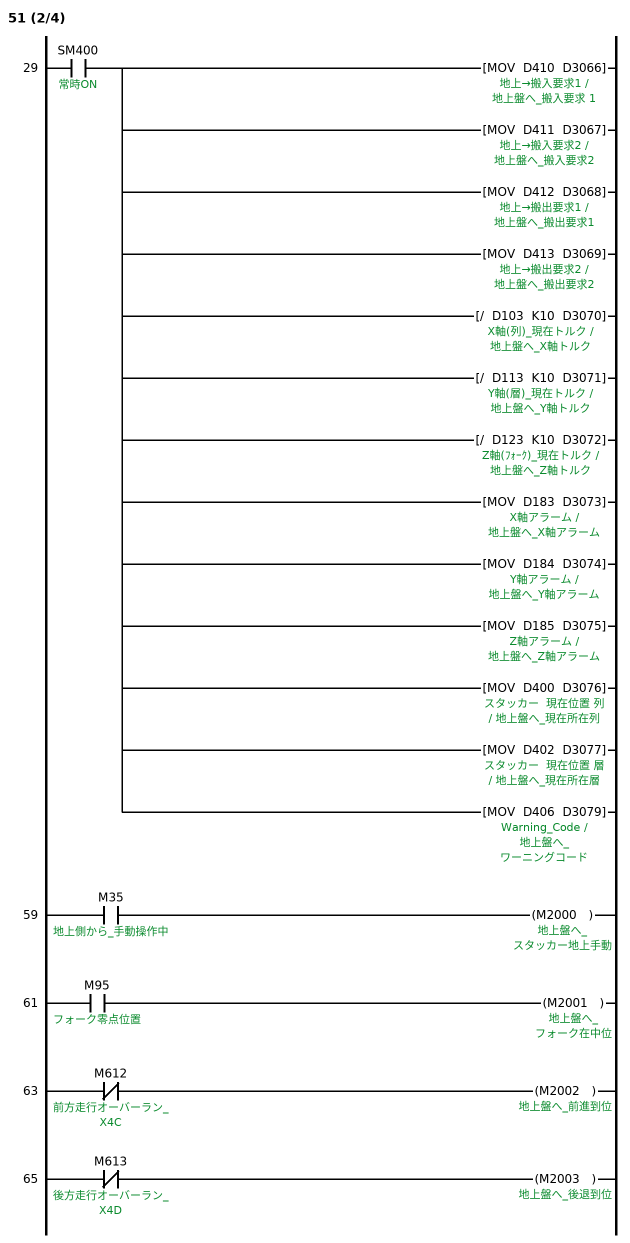
29    LD      SM400  ; 常時ON
      MOV     D410 D3066  ; 地上→搬入要求1 / 地上盤へ_搬入要求 1
      MOV     D411 D3067  ; 地上→搬入要求2 / 地上盤へ_搬入要求2
      MOV     D412 D3068  ; 地上→搬出要求1 / 地上盤へ_搬出要求1
      MOV     D413 D3069  ; 地上→搬出要求2 / 地上盤へ_搬出要求2
      /       D103 K10 D3070  ; X軸(列)_現在トルク / 地上盤へ_X軸トルク
      /       D113 K10 D3071  ; Y軸(層)_現在トルク / 地上盤へ_Y軸トルク
      /       D123 K10 D3072  ; Z軸(ﾌｫｰｸ)_現在トルク / 地上盤へ_Z軸トルク
      MOV     D183 D3073  ; X軸アラーム / 地上盤へ_X軸アラーム
      MOV     D184 D3074  ; Y軸アラーム / 地上盤へ_Y軸アラーム
      MOV     D185 D3075  ; Z軸アラーム / 地上盤へ_Z軸アラーム
      MOV     D400 D3076  ; スタッカー  現在位置 列 / 地上盤へ_現在所在列
      MOV     D402 D3077  ; スタッカー  現在位置 層 / 地上盤へ_現在所在層
      MOV     D406 D3079  ; Warning_Code / 地上盤へ_ワーニングコード
59    LD      M35  ; 地上側から_手動操作中
      OUT     M2000  ; 地上盤へ_スタッカー地上手動
61    LD      M95  ; フォーク零点位置
      OUT     M2001  ; 地上盤へ_フォーク在中位
63    LDI     M612  ; 前方走行オーバーラン_X4C
      OUT     M2002  ; 地上盤へ_前進到位
65    LDI     M613  ; 後方走行オーバーラン_X4D
      OUT     M2003  ; 地上盤へ_後退到位
